TYPE "PLCtoMES_SubCheckIn_ext"
VERSION : 0.1
   STRUCT
      Load_SubPart1ChickInReq : Bool;
      Load_SubPart2ChickInReq : Bool;
      Load_SubPart3ChickInReq : Bool;
      Load_SubPart4ChickInReq : Bool;
      Load_SubPart5ChickInReq : Bool;
      Load_SubPart6ChickInReq : Bool;
      Load_SubPart7ChickInReq : Bool;
      Load_SubPart8ChickInReq : Bool;
   END_STRUCT;

END_TYPE

